FUNCTION_BLOCK ProcessStep EXTENDS SM_ProcessStep
VAR_INPUT
    description : STRING;
END_VAR
VAR_OUTPUT
END_VAR
VAR
END_VAR

SUPER^(process := process);

METHOD isGood : BOOL
VAR_INPUT
END_VAR
isGood := process.isGood();
END_METHOD

METHOD isWarning : BOOL
VAR_INPUT
END_VAR
isWarning := process.statuses.healthStatus.warning;
END_METHOD

METHOD isBusy : BOOL
VAR_INPUT
END_VAR
isBusy := process.isBusy();
END_METHOD

METHOD PUBLIC isBad : BOOL
VAR_INPUT
END_VAR
isBad := process.statuses.healthStatus.bad;
END_METHOD

END_FUNCTION_BLOCK

(* stored: Version 1.1.0.1, ProductVersion 3.1.4018.5
   POU ProcessStep: Id {7c51619e-83d4-46a7-a398-0a62ddb01b00}, SpecialFunc None
   Method isGood: Id {3544d4be-a81a-40e4-b766-2f6f4ab94c30}
   Method isWarning: Id {4dee5d8d-a7e5-4b7a-bffa-fb3edf3a20bb}
   Method isBusy: Id {50ed5c86-eef4-47fb-8be0-ca8763849513}
   Method isBad: Id {df13a064-fda5-4465-9f5e-fb9e93b506a6} *)
